{attribute 'qualified_only'}
{attribute 'strict'}
{attribute 'to_string'}
TYPE E_MoveDoneCause :
(
    UNKNOWN := 0,           // DEFAULT/UNCATEGORIZED
    MOVEDONE,               // ABSOLUTE MOVE COMPLETED
    STEPMOVEDONE,           // STEP/JOG MOVE COMPLETED
    HOMEDONE,               // HOMING COMPLETED
    CALIBRATIONDONE,        // CALIBRATION COMPLETED
    RESETDONE,              // RESET COMMAND COMPLETED
    HALTDONE,               // MANUAL HALT COMPLETED
    ABORTEDHOME,            // HOME ABORTED
    ABORTEDSTEPMOVE,        // STEP MOVE ABORTED
    ABORTEDCALIBRATION,     // CALIBRATION ABORTED
    REFERENCED,             // AXIS BECAME REFERENCED
    CALIBRATED              // AXIS BECAME CALIBRATED
);
END_TYPE

(* stored: Version 1.1.0.1
   DUT E_MoveDoneCause: Id {f11d0b8d-a319-4919-8ad2-0dfa2b932888} *)
